# B&R Automation Studio project MirrElszkowskischody
Automation Studio 3.0.90.38 SP20; Default project

## Configuration 4PP481

### Task classes (Cpu.sw)
```
Cyclic#4:
  Tunel <- Tunel.prg
Libraries: standard
```

### IoMap.iom - PLC1/IoMap.iom
```iecst
(********************************************************************
 * COPYRIGHT --
 ********************************************************************
 * File: IoMap.iom
 * Author: User
 * Created: November 09, 2017
 ********************************************************************
 * IO mapping file
 ********************************************************************)
VAR_CONFIG
	Tunel.Tunel.diStart AT %IX.SL1.SS1.IF1.ST2.DigitalInput01;
	Tunel.Tunel.diStop AT %IX.SL1.SS1.IF1.ST2.DigitalInput02;
	Tunel.Tunel.diEStop AT %IX.SL1.SS1.IF1.ST2.DigitalInput03;
	Tunel.Tunel.diCzujnikSpalin1 AT %IX.SL1.SS1.IF1.ST2.DigitalInput04;
	Tunel.Tunel.diCzujnikSpalin2 AT %IX.SL1.SS1.IF1.ST2.DigitalInput05;
	Tunel.Tunel.diCzujnikSpalin3 AT %IX.SL1.SS1.IF1.ST2.DigitalInput06;
	Tunel.Tunel.doSystemAktywny AT %QX.SL1.SS1.IF1.ST3.DigitalOutput01;
	Tunel.Tunel.doWentylatorM1 AT %QX.SL1.SS1.IF1.ST3.DigitalOutput02;
	Tunel.Tunel.doWentylatorM2 AT %QX.SL1.SS1.IF1.ST3.DigitalOutput03;
	Tunel.Tunel.doWentylatorM3 AT %QX.SL1.SS1.IF1.ST3.DigitalOutput04;
	Tunel.Tunel.diCzujnikSpalin4 AT %IX.SL1.SS1.IF1.ST2.DigitalInput07;
END_VAR
```

## Configuration Simulation

### Task classes (Cpu.sw)
```
Cyclic#4:
  Tunel <- Tunel.prg
Libraries: AsIecCon, astime, standard
```

## Logical view

Binary libraries used (declarations not repeated): astime, OPERATOR, standard

### Package Logical/Libraries - Global libraries

- Visualisation Logical/Visu (not shown)

### Program Logical/Tunel (IEC) - A new program

#### TunelCyclic.ab - Cyclic code
```automation-basic
(********************************************************************
 * COPYRIGHT --
 ********************************************************************
 * Program: Tunel
 * File: TunelCyclic.ab
 * Author: Liss_1
 * Created: January 25, 2018
 ********************************************************************
 * Implementation of program Tunel
 ********************************************************************)

PROGRAM _CYCLIC

	Tunel.doSystemAktywny = ( (Tunel.diStart OR Tunel.doSystemAktywny) AND NOT (Tunel.diStop) )
	Tunel.doSystemAktywny = Tunel.doSystemAktywny AND Tunel.diEStop
	IF (Tunel.doSystemAktywny = FALSE) THEN

		Tunel.doWentylatorM1 = FALSE
		Tunel.doWentylatorM2 = FALSE
		Tunel.doWentylatorM3 = FALSE
	ELSE
		Tunel.doWentylatorM1 = Tunel.diCzujnikSpalin1 AND Tunel.diCzujnikSpalin2
		Tunel.doWentylatorM2 = Tunel.diCzujnikSpalin2 AND Tunel.diCzujnikSpalin3
		Tunel.doWentylatorM3 = Tunel.diCzujnikSpalin3 AND Tunel.diCzujnikSpalin4

	ENDIF

END_PROGRAM
```

#### TunelInit.ab - Initialization code
```automation-basic
(********************************************************************
 * COPYRIGHT --
 ********************************************************************
 * PROGRAM: Tunel
 * File: TunelInit.ab
 * Author: Liss_1
 * Created: January 25, 2018
 ********************************************************************
 * Implementation OF PROGRAM Tunel
 ********************************************************************)

PROGRAM _INIT

(* TODO : Add your code here *)

END_PROGRAM
```

#### Tunel.typ - Local data types
```iecst
(********************************************************************
 * COPYRIGHT --
 ********************************************************************
 * Program: TunelPROGRAM
 * File: TunelPROGRAM.typ
 * Author: pmizo
 * Created: January 18, 2018
 ********************************************************************
 * Local data types of program TunelPROGRAM
 ********************************************************************)

TYPE
	TunelStruct : 	STRUCT
		diCzujnikSpalin1 : BOOL := FALSE;
		diCzujnikSpalin2 : BOOL := FALSE;
		diCzujnikSpalin3 : BOOL := FALSE;
		diCzujnikSpalin4 : BOOL := FALSE;
		diEStop : BOOL := TRUE;
		diStart : BOOL := FALSE;
		diStop : BOOL := FALSE;
		doSystemAktywny : BOOL := FALSE;
		doWentylatorM3 : BOOL := FALSE;
		doWentylatorM2 : BOOL := FALSE;
		doWentylatorM1 : BOOL := FALSE;
	END_STRUCT;
END_TYPE
```

#### Tunel.var - Local variables
```iecst
(********************************************************************
 * COPYRIGHT --
 ********************************************************************
 * Program: TunelPROGRAM
 * File: TunelPROGRAM.var
 * Author: pmizo
 * Created: January 18, 2018
 ********************************************************************
 * Local variables of program TunelPROGRAM
 ********************************************************************)
VAR
	Tunel : TunelStruct;
END_VAR
```

### Program Logical/Ppoz

#### Ppoz.typ
```iecst
(********************************************************************
 * COPYRIGHT --
 ********************************************************************
 * Program: Ppoz
 * File: Ppoz.typ
 * Author: User
 * Created: November 16, 2017
 ********************************************************************
 * Local data types of program Ppoz
 ********************************************************************)

TYPE
	SystemStruct : 	STRUCT
		diStop : BOOL;
		diStart : BOOL;
		uiStop : BOOL;
		uiStart : BOOL;
		uiSystemAktywny : BOOL;
		doSystemAktywny : BOOL;
		diReset : BOOL;
		uiReset : BOOL;
		doSyrena : BOOL;
		uiSyrena : BOOL;
		doKogut : BOOL;
		uiKogut : BOOL;
	END_STRUCT;
	RoomStruct : 	STRUCT
		uiCzujnikSwiatlo : BOOL;
		uiCzujnikTemp : BOOL;
		uiTryskacz : BOOL;
		uiCzujnikDym : BOOL;
		diCzujnikSwiatlo : BOOL;
		diCzujnikTemp : BOOL;
		doTryskacz : BOOL;
		diCzujnikDym : BOOL;
	END_STRUCT;
END_TYPE
```

#### Ppoz.var
```iecst
(********************************************************************
 * COPYRIGHT --
 ********************************************************************
 * Program: Ppoz
 * File: Ppoz.var
 * Author: User
 * Created: November 16, 2017
 ********************************************************************
 * Local variables of program Ppoz
 ********************************************************************)
VAR
	System : SystemStruct;
	Room : ARRAY[0..9] OF RoomStruct := [10(0)];
	uiModeWork : USINT := 0;
	flagaView : INT;
END_VAR
```

#### Ppoz.ab
```automation-basic
(********************************************************************
 * COPYRIGHT --
 ********************************************************************
 * Program: Ppoz
 * File: Ppoz.ab
 * Author: User
 * Created: November 16, 2017
 ********************************************************************
 * Implementation of program Ppoz
 ********************************************************************)

PROGRAM _INIT
	flagaView = 0

	uiModeWork = 2

END_PROGRAM

PROGRAM _CYCLIC
	CASE uiModeWork OF
		ACTION 1:
			Room[0].doTryskacz = Room[0].uiTryskacz
			System.doKogut = System.uiKogut
			System.doSyrena = System.uiSyrena
			ENDACTION
		ACTION 2:
			System.doSystemAktywny = (((System.diStart OR System.uiStart) OR System.doSystemAktywny) AND (NOT(System.diStop) OR NOT (System.uiStop)))
			IF System.doSystemAktywny THEN
				Room[0].doTryskacz = (Room[0].diCzujnikDym AND Room[0].diCzujnikSwiatlo AND NOT (Room[0].diCzujnikTemp)) OR  \
				(Room[0].diCzujnikDym AND NOT (Room[0].diCzujnikSwiatlo) AND Room[0].diCzujnikTemp) OR \
				(NOT (Room[0].diCzujnikDym) AND Room[0].diCzujnikSwiatlo AND Room[0].diCzujnikTemp) OR \
				(Room[0].diCzujnikDym AND Room[0].diCzujnikSwiatlo AND Room[0].diCzujnikTemp)
					System.doSyrena = Room[0].doTryskacz AND NOT(System.diReset)
					System.doKogut = Room[0].doTryskacz
				ELSE
					Room[0].doTryskacz = FALSE
					System.doSyrena = FALSE
					System.doKogut = FALSE

				ENDIF
		ENDACTION
ENDCASE
END_PROGRAM

PROGRAM _EXIT

(* TODO : Add your code here *)

END_PROGRAM
```

- Program Logical/schody (IEC) (no source held here)

### Program Logical/Tunel - Kopia (IEC)

#### Tunel.ab - Implementation code
```automation-basic
(********************************************************************
 * COPYRIGHT -- Microsoft
 ********************************************************************
 * Program: Tunel
 * File: Tunel.ab
 * Author: Liss_1
 * Created: January 25, 2018
 ********************************************************************
 * Implementation of program Tunel
 ********************************************************************)

PROGRAM _INIT

(* TODO : Add your code here *)

END_PROGRAM

PROGRAM _CYCLIC

(* TODO : Add your code here *)

END_PROGRAM

PROGRAM _EXIT

(* TODO : Add your code here *)

END_PROGRAM
```

### Zarowa.var
```iecst
(********************************************************************
 * COPYRIGHT --
 ********************************************************************
 * Program: Zarowa
 * File: Zarowa.var
 * Author: User
 * Created: November 09, 2017
 ********************************************************************
 * Local variables of program Zarowa
 ********************************************************************)
VAR
	doZarowka : ARRAY[0..9] OF BOOL;
	diPrzelacznik : ARRAY[0..9] OF BOOL;
END_VAR
```

### Program Logical/Zarowa_b

#### Zarowa.ab
```automation-basic
(********************************************************************
 * COPYRIGHT --
 ********************************************************************
 * Program: Zarowa
 * File: Zarowa.ab
 * Author: User
 * Created: November 09, 2017
 ********************************************************************
 * Implementation of program Zarowa
 ********************************************************************)

PROGRAM _INIT

(* TODO : Add your code here *)

END_PROGRAM

PROGRAM _CYCLIC

	doZarowka[0] = diPrzelacznik[0]

END_PROGRAM

PROGRAM _EXIT

(* TODO : Add your code here *)

END_PROGRAM
```

Listed in the project but not available here: Logical/Global.typ, Logical/schody/schody.ab, Logical/schody/schody.var
